PROGRAM Pneumatics_Template
VAR
END_VAR

//Set initial parameters:

(*
stPneumaticAxisStruct.stPneumaticAxisInputs.bPermit := TRUE (to enable cylinder to move)
If stPneumaticAxisStruct.stPneumaticAxisInputs.bPermit is not set to true before going online, error will appear.
Set stPneumaticAxisStruct.stPneumaticAxisInputs.bPermit := TRUE, and reset errors with E_PneumaticMode.RESET.

Select the wanted mode of work.
Default state is E_PneumaticMode.SINGLE_SOLENOID_PLC.

For E_PneumaticMode.SINGLE_SOLENOID_PLC:

Define:
nTimeToExtract and nTimeToRetract in seconds (if you want the time to be 10s just write 10)
It’s assumed that the cylinder is retracted and the bLimitBackward is activated:
Set stPneumaticAxisStruct.stPneumaticAxisInputs.bLimitBwd := TRUE

To start extraction: stPneumaticAxisStruct.stPneumaticAxisControl.bStartExtend := TRUE;
This will activate the timing of the command, with fbTimerStartMoving.
Set stPneumaticAxisStruct.stPneumaticAxisInputs.bLimitBwd := FALSE, to simulate cylider moving
If the stPneumaticAxisStruct.stPneumaticAxisInputs.bLimitFwd is not deactivated in given time (it's set to 10s by default), it’s assumed that the cylinder has not moved and this will cause it to go to the error state.
If the end position is not reached within time defined in nTimeToExtract, the system will show error.
Set stPneumaticAxisStruct.stPneumaticAxisInputs.bLimitFwd := TRUE (to simulate finishing of extraction)

To reset errors, change state to  E_PneumaticMode.RESET.

To move cylinder backwards: stPneumaticAxisStruct.stPneumaticAxisControl.bStartRetract := TRUE;
Set stPneumaticAxisStruct.stPneumaticAxisInputs.bLimitFwd := FALSE;
The cylinder is retracted when stPneumaticAxisStruct.stPneumaticAxisInputs.bLimitBwd := TRUE (you have to make it TRUE manually to simulate the finish of the moving).
If this doesn’t happen in specified time, in nTimeToRetract, state machine goes into error state.

To reset errors, change state to  E_PneumaticMode.RESET.

For E_PneumaticMode.SINGLE_SOLENOID_MANUAL:

Same prinicples apply, control is done with two signals:
stPneumaticAxisStruct.stPneumaticAxisInputs.bExtendCylinderManual := TRUE to extract cylinder
stPneumaticAxisStruct.stPneumaticAxisInputs.bRetractCylinderManual := TRUE to retract cylinder

RS function blocks are used to handle signals from the extend/retract push buttons.

Reset errors with E_PneumaticMode.RESET

*)

END_PROGRAM

(* stored: Version 1.1.0.1, ProductVersion 3.1.4024.5
   POU Pneumatics_Template: Id {7bf401fb-a600-4741-a67b-36f20e194cfc}, SpecialFunc None *)
